RoboDK station: tarea2_isabellaceballos.rdk

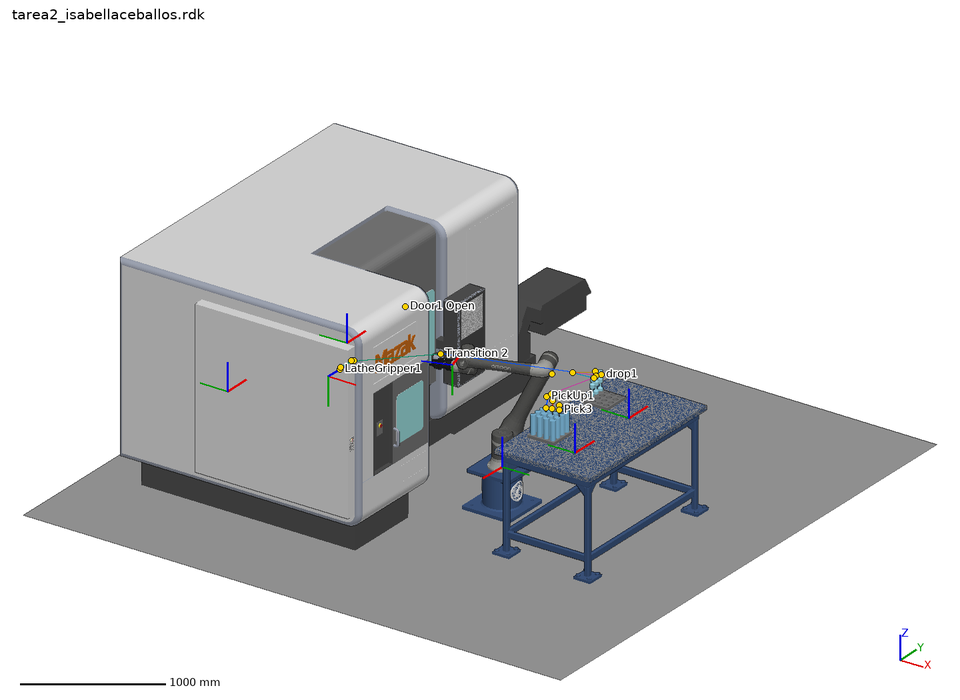
[picture v0: the station drawn from its stored meshes, robots at their saved joint values, targets as dots, program paths as lines]
Station tarea2_isabellaceballos (saved by RoboDK 5.5.1). Poses are relative to the parent item; angles as X-Y-Z fixed-axis rotations.
Station parameters (name, value as stored): TAGS, ['Machine Tending', 'CNC']
  - frame Omron TM12X Base at (300, 0, 70) mm, rotated rx 0 ry 0 rz -90 deg
    - robot Omron TM12X: 6 axes, payload 12 kg, reach 1300 mm, repeatability 0.1 mm, weight 33.3 kg
        modified DH rows (alpha deg, a mm, theta deg, d mm): 0, 0, 0, 165.2; 90, 0, 90, 0; 0, 636.1, 0, 0; 0, 557.9, -90, 156.3; -90, 0, 0, 106; 90, 0, 180, 113.15
        joint limits [-360, -360, -163, -360, -360, -360] to [360, 360, 163, 360, 360, 360]; home [0, 0, 90, -90, 90, 0]; saved at [291.3, -25.7, 113.76, -268.05, -85.72, 0]
      - frame RobotiQ HandE Dual Gripper at (0, 0, -5) mm
      - tool RobotiQ 2F-85 Gripper (Closed), TCP at (0, 0, 130) mm, size 134.4 x 157.6 x 75 mm
    - object Pedestal H12in (Type 1) at (0, 0, -300) mm, size 400 x 400 x 304.8 mm, geometry from Pedestal-H12in-Type-1.sld
  - frame Mazak Lathe Base at (-1000, 0, 650) mm, rotated rx 0 ry 0 rz 90 deg
    - frame Lathe at (-368.68, -104.77, -79.13) mm, rotated rx -90 ry 0 rz -90 deg
      - target LatheGripper1 (Cartesian target) at (-0.18, 0.1, 134.88) mm, rotated rx 0 ry 90 rz 165 deg; joints [296.712, 22.07, 84.693, -319.639, -67.09, 75.877] of Omron TM12X
      - target App1LatheGripper2 (Cartesian target) at (-0.18, 0.1, 301.9) mm, rotated rx 0 ry 90 rz 165 deg; joints [285.755, 19.624, 87.976, -318.559, -76.4, 81.971] of Omron TM12X
      - target App1LatheGripper (Cartesian target) at (-2.45, -8.35, 278.24) mm, rotated rx -90 ry -0.7 rz 75 deg; joints [284.667, 42.036, 44.196, -250.751, -75.843, 93.179] of Omron TM12X
      - target LatheGripper (Cartesian target) at (-2.58, -8.82, 147.35) mm, rotated rx -90 ry -0.7 rz 75 deg; joints [292.046, 45.075, 38.746, -247.697, -68.742, 95.287] of Omron TM12X
    - robot Mazak Lathe: 1 axes
        modified DH rows (alpha deg, a mm, theta deg, d mm): 0, 0, 0, 0 linear
        base shift (0, 0, 0) mm, rotated rx 0 ry 90 rz 0 deg
        joint limits [0] to [700]; home [0]; saved at [0]
  - frame Input at (1200, -410, 590) mm, rotated rx 0 ry 0 rz 90 deg
    - object Part Matrix at (0, 180, 30) mm, size 220 x 220 x 25 mm, geometry from Part Matrix.step
    - object Part 16 at (27.5, 207.5, 30) mm, size 40 x 40 x 150 mm, geometry from Part.step
    - object Part 15 at (27.5, 262.5, 30) mm, size 40 x 40 x 150 mm, geometry from Part.step
    - object Part 14 at (27.5, 317.5, 30) mm, size 40 x 40 x 150 mm, geometry from Part.step
    - object Part 12 at (82.5, 207.5, 30) mm, size 40 x 40 x 150 mm, geometry from Part.step
    - object Part 11 at (82.5, 262.5, 30) mm, size 40 x 40 x 150 mm, geometry from Part.step
    - object Part 10 at (82.5, 317.5, 30) mm, size 40 x 40 x 150 mm, geometry from Part.step
    - object Part 9 at (82.5, 372.5, 30) mm, size 40 x 40 x 150 mm, geometry from Part.step
    - object Part 8 at (137.5, 207.5, 30) mm, size 40 x 40 x 150 mm, geometry from Part.step
    - object Part 6 at (137.5, 317.5, 30) mm, size 40 x 40 x 150 mm, geometry from Part.step
    - object Part Done 16 at (27.5, 27.5, -20) mm, size 40.5 x 40.5 x 150 mm, geometry from Part Done.step
    - object Part Done 15 at (27.5, 82.5, -20) mm, size 40.5 x 40.5 x 150 mm, geometry from Part Done.step
    - object Part Done 14 at (27.5, 137.5, -20) mm, size 40.5 x 40.5 x 150 mm, geometry from Part Done.step
    - object Part Done 13 at (27.5, 192.5, -20) mm, size 40.5 x 40.5 x 150 mm, geometry from Part Done.step
    - object Part Done 12 at (82.5, 27.5, -20) mm, size 40.5 x 40.5 x 150 mm, geometry from Part Done.step
    - object Part Done 11 at (82.5, 82.5, -20) mm, size 40.5 x 40.5 x 150 mm, geometry from Part Done.step
    - object Part Done 10 at (82.5, 137.5, -20) mm, size 40.5 x 40.5 x 150 mm, geometry from Part Done.step
    - object Part Done 9 at (82.5, 192.5, -20) mm, size 40.5 x 40.5 x 150 mm, geometry from Part Done.step
    - object Part Done 8 at (137.5, 27.5, -20) mm, size 40.5 x 40.5 x 150 mm, geometry from Part Done.step
    - object Part Done 7 at (137.5, 82.5, -20) mm, size 40.5 x 40.5 x 150 mm, geometry from Part Done.step
    - object Part Done 6 at (137.5, 137.5, -20) mm, size 40.5 x 40.5 x 150 mm, geometry from Part Done.step
    - object Part Done 5 at (137.5, 192.5, -20) mm, size 40.5 x 40.5 x 150 mm, geometry from Part Done.step
    - object Part 7 at (137.5, 262.5, 30) mm, size 40 x 40 x 150 mm, geometry from Part.step
    - object Part 4 at (192.5, 207.5, 30) mm, rotated rx 0 ry 0 rz -180 deg, size 40 x 40 x 150 mm, geometry from Part.step
    - object Part Done 4 at (192.5, 27.5, -20) mm, rotated rx 0 ry 0 rz 180 deg, size 40.5 x 40.5 x 150 mm, geometry from Part Done.step
    - object Part 13 at (27.5, 372.5, 30) mm, size 40 x 40 x 150 mm, geometry from Part.step
    - target PickUp1 (Cartesian target) at (197.79, 377.57, 243.21) mm, rotated rx -90.01 ry 0 rz -179.05 deg; joints [78.517, -21.194, 99.72, -258.517, -102.431, -0.005] of Omron TM12X
    - target Pick1 (Cartesian target) at (192.26, 377.49, 159.76) mm, rotated rx -90.01 ry 0 rz -179.05 deg; joints [77.548, -21.82, 108.73, -266.901, -103.4, -0.006] of Omron TM12X
    - object Part 5 at (137.5, 372.5, 30) mm, size 40 x 40 x 150 mm, geometry from Part.step
    - target PickUp2 (Cartesian target) at (201.47, 332.43, 224.78) mm, rotated rx -90 ry 3.89 rz 135.95 deg; joints [107.585, -17.36, 99.274, -261.904, -28.363, 3.902] of Omron TM12X
    - target Pick2 (Cartesian target) at (194.9, 329.64, 168.72) mm, rotated rx -90 ry 3.89 rz 135.95 deg; joints [106.47, -17.482, 105.138, -267.647, -29.478, 3.901] of Omron TM12X
    - target PickUp3 (Cartesian target) at (198, 272.34, 206.6) mm, rotated rx -90.01 ry -0.01 rz 147.63 deg; joints [100.342, -14.09, 98.9, -264.802, -47.286, -0.002] of Omron TM12X
    - target Pick3 (Cartesian target) at (197.73, 271.91, 171.16) mm, rotated rx -90.01 ry -0.01 rz 147.63 deg; joints [100.293, -14.235, 102.652, -268.408, -47.336, -0.002] of Omron TM12X
  - frame Output at (1200, 230, 600) mm, rotated rx 0 ry 0 rz 90 deg
    - object Part Matrix at (0, 180, 30) mm, size 220 x 220 x 25 mm, geometry from Part Matrix.step
      - object Part 1 at (193.5, 178.91, -12.21) mm, rotated rx 0 ry -0.01 rz -111.33 deg, size 40 x 40 x 150 mm, geometry from Part.step
      - object Part Done 1 at (191.78, 194.55, 1.25) mm, rotated rx -0.18 ry -0.67 rz -15.38 deg, size 40.5 x 40.5 x 150 mm, geometry from Part Done.step
      - object Part 2 at (150.87, 185.46, -11.65) mm, rotated rx -2.71 ry -2.79 rz -101.16 deg, size 40 x 40 x 150 mm, geometry from Part.step
      - object Part Done 2 at (138.14, 192.48, 0.91) mm, rotated rx -0.17 ry -0.68 rz 49.72 deg, size 40.5 x 40.5 x 150 mm, geometry from Part Done.step
      - object Part 3 at (93.46, 178.8, -3.24) mm, rotated rx -4.21 ry 0.62 rz -139.81 deg, size 40 x 40 x 150 mm, geometry from Part.step
      - object Part Done 3 at (82.22, 190.38, 2.81) mm, rotated rx 4.03 ry 0 rz 22.82 deg, size 40.5 x 40.5 x 150 mm, geometry from Part Done.step
    - target drop1 (Cartesian target) at (198.5, 367.59, 147.55) mm, rotated rx -90 ry 0 rz 149.62 deg; joints [163.829, 5.576, 85.939, -271.515, 14.209, 0] of Omron TM12X
    - target UpDrop2 (Cartesian target) at (147.69, 382.37, 191.36) mm, rotated rx -90.01 ry 0 rz -145.27 deg; joints [150.104, -17.325, 101.671, -264.336, -64.625, 0.007] of Omron TM12X
    - target Drop2 (Cartesian target) at (147.19, 375.55, 157.21) mm, rotated rx -90.01 ry 0 rz -145.27 deg; joints [149.15, -17.018, 104.984, -267.956, -65.579, 0.007] of Omron TM12X
    - target Drop3 (Cartesian target) at (96.91, 360.44, 168.27) mm, rotated rx -93.89 ry -1.74 rz -172.1 deg; joints [156.377, -14.102, 122.108, -100.567, 31.62, 184.605] of Omron TM12X
  - frame World at (-2000, 0, 0) mm, rotated rx 0 ry 0 rz 90 deg
    - target Door1 Open (Cartesian target) at (700, -1000, 650) mm; joints [700, 0, 0, 0, 0, 0]
    - target Door1 Close (Cartesian target) at (0, -1000, 650) mm; joints [0, 0, 0, 0, 0, 0] of Mazak Lathe
    - object Floor at (250, -1940, -230) mm, size 4500 x 4500 x 0 mm, geometry from Floor (2).sld
    - object Table 1400x800x800mm at (-340, -3110, 590) mm, size 1420 x 820 x 800 mm, geometry from Table-1400x800x800mm.sld
    - target Home (Cartesian target) at (-159.05, -2821.45, 833.21) mm, rotated rx 0 ry 90 rz -134.05 deg; joints [118.439, -21.833, 100.089, -258.241, -17.509, 90.005] of Omron TM12X
    - target Transition1 (Cartesian target) at (332.55, -2486.73, 697.08) mm, rotated rx -89.14 ry -2.2 rz -141.74 deg; joints [240.5, -44.888, 123.151, -255.991, 22.223, -0.096] of Omron TM12X
    - target trans1 (Cartesian target) at (201.2, -2749.5, 833.2) mm, rotated rx 0 ry 90 rz -78.57 deg; joints [162.747, -30.859, 104.408, -253.528, -28.687, 90.017] of Omron TM12X
    - target Target 6 (Cartesian target) at (-159.05, -2821.45, 833.21) mm, rotated rx -116.03 ry 89.99 rz 109.92 deg; joints [120.666, -29.131, 103.705, -254.562, -60.282, 0.002] of Omron TM12X
    - target Transition 2 (joint target) at (110.77, -1705.81, 721.22) mm, rotated rx -130.72 ry 89.99 rz -68.7 deg; joints [291.3, -25.7, 113.76, -268.05, -85.72, 0]
    - target DOOROPEN (Cartesian target) at (700, -1000, 650) mm; joints [700] of Mazak Lathe
    - target DOOR CLOSE (Cartesian target) at (0, -1000, 650) mm; joints [0] of Mazak Lathe
    - target Target 10 (joint target) at (0, -1000, 650) mm; joints [0] of Mazak Lathe
  - folder Mechanism Programs
    - program OpenDoor1 (1 instructions, listed below)
    - program CloseDoor1 (1 instructions, listed below)
  - folder PickInput Programs
    - program Pick 1 (6 instructions, listed below)
    - program Pick 2 (6 instructions, listed below)
    - program Pick 3 (6 instructions, listed below)
  - folder DropOutput Programs
    - program Drop 1 (9 instructions, listed below)
    - program Drop 2 (8 instructions, listed below)
    - program Drop 3 (7 instructions, listed below)
  - folder Other Programs
    - program GoHome (3 instructions, listed below)
    - program ReplaceObjects (1 instructions, listed below)
    - program Init (6 instructions, listed below)
    - program PickLatheTransition (4 instructions, listed below)
  - folder Lath Programs
    - folder Work Programs
      - program Work 1 (3 instructions, listed below)
      - program Work 2 (3 instructions, listed below)
      - program Work 3 (3 instructions, listed below)
    - program PickLathe (11 instructions, listed below)
    - program DropLathe (10 instructions, listed below)
  - program Reset (2 instructions, listed below)
  - program MainProgram2 (22 instructions, listed below)
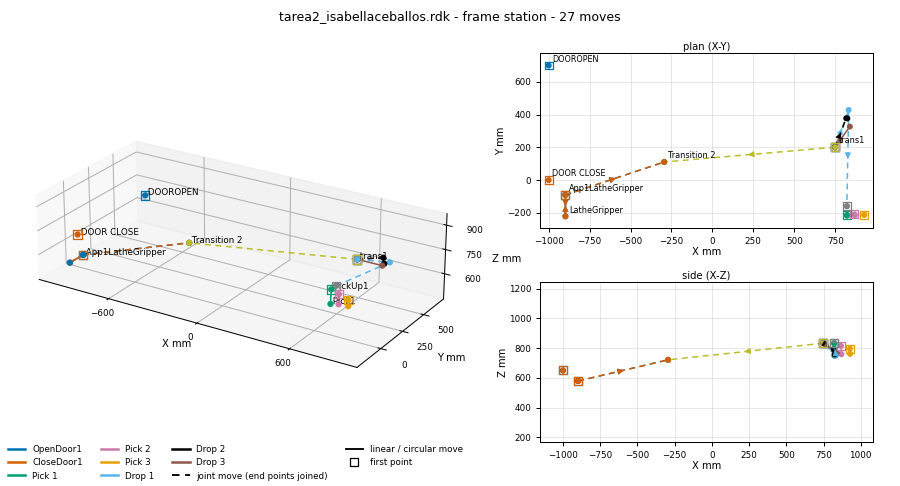
[picture p0: tool path of tarea2_isabellaceballos.rdk in frame station, 27 of 27 moves have a stored position in this frame; points joined in program order, loops and branches not executed]

--- program OpenDoor1 (robot Mazak Lathe) ---
  MoveJ (DOOROPEN)

--- program CloseDoor1 (robot Mazak Lathe) ---
  MoveJ (DOOR CLOSE)

--- program Pick 1 (robot Omron TM12X) ---
  Set Ref.: Input
  Est. herr: RobotiQ 2F-85 Gripper (Closed)
  MoveJ (PickUp1)
  MoveL (Pick1)
  Adjuntar a RobotiQ 2F-85 Gripper (Closed)
  Llamar GoHome

--- program Pick 2 (robot Omron TM12X) ---
  Set Ref.: Input
  Est. herr: RobotiQ 2F-85 Gripper (Closed)
  MoveJ (PickUp2)
  MoveL (Pick2)
  Adjuntar a RobotiQ 2F-85 Gripper (Closed)
  Llamar GoHome

--- program Pick 3 (robot Omron TM12X) ---
  Set Ref.: Input
  Est. herr: RobotiQ 2F-85 Gripper (Closed)
  MoveJ (PickUp3)
  MoveL (Pick3)
  Adjuntar a RobotiQ 2F-85 Gripper (Closed)
  Llamar GoHome

--- program Drop 1 (robot Omron TM12X) ---
  Set Ref.: World
  Est. herr: RobotiQ 2F-85 Gripper (Closed)
  MoveJ (trans1)
  Set Ref.: Output
  Est. herr: RobotiQ 2F-85 Gripper (Closed)
  MoveJ (drop1)
  Separar de RobotiQ 2F-85 Gripper (Closed)
  Set Ref.: World
  MoveJ (Home)

--- program Drop 2 (robot Omron TM12X) ---
  Set Ref.: World
  MoveJ (trans1)
  Set Ref.: Output
  Est. herr: RobotiQ 2F-85 Gripper (Closed)
  MoveJ (UpDrop2)
  MoveL (Drop2)
  Separar de RobotiQ 2F-85 Gripper (Closed)
  Llamar GoHome

--- program Drop 3 (robot Omron TM12X) ---
  Set Ref.: World
  MoveJ (trans1)
  Set Ref.: Output
  Est. herr: RobotiQ 2F-85 Gripper (Closed)
  MoveL (Target 4) -> target Drop3
  Separar de RobotiQ 2F-85 Gripper (Closed)
  Llamar GoHome

--- program GoHome (robot Omron TM12X) ---
  Set Ref.: World
  Set Tool: Gripper1 at (145, 0, 130) mm, rotated rx 45 ry 0 rz 90 deg
  MoveJ (Home)

--- program ReplaceObjects (robot Omron TM12X) ---
  Reemplazar objetos

--- program Init (robot Omron TM12X) ---
  Run OpenGripper1
  Run OpenGripper2
  Run CloseDoor1
  Run ReplaceObjects
  Show objects
  Hide objects

--- program PickLatheTransition (robot Omron TM12X) ---
  Set Ref.: World
  Set Tool: Gripper1 at (145, 0, 130) mm, rotated rx 45 ry 0 rz 90 deg
  MoveJ (trans1)
  MoveJ (Transition 2)

--- program Work 1 (robot Omron TM12X) ---
  Pausa 3.0 s
  Mostrar Part Done 1
  Hide Part 1

--- program Work 2 (robot Omron TM12X) ---
  Pausa 3.0 s
  Show Part Done 2
  Hide Part 2

--- program Work 3 (robot Omron TM12X) ---
  Pausa 3.0 s
  Show Part Done 3
  Hide Part 3

--- program PickLathe (robot Omron TM12X) ---
  Set Ref.: Lathe
  Est. herr: RobotiQ 2F-85 Gripper (Closed)
  Llamar OpenDoor1
  MoveJ (App1LatheGripper)
  MoveL (LatheGripper)
  Adjuntar a RobotiQ 2F-85 Gripper (Closed)
  Adjuntar a RobotiQ 2F-85 Gripper (Closed)
  MoveJ (App1LatheGripper)
  Set Ref.: World
  MoveJ (Transition 2)
  Llamar CloseDoor1

--- program DropLathe (robot Omron TM12X) ---
  Set Ref.: Lathe
  Est. herr: RobotiQ 2F-85 Gripper (Closed)
  Llamar OpenDoor1
  MoveJ (App1LatheGripper1)
  MoveL (LatheGripper)
  Separar de RobotiQ 2F-85 Gripper (Closed)
  MoveJ (App1LatheGripper1)
  Set Ref.: World
  MoveJ (Transition 2)
  Llamar CloseDoor1

--- program Reset (robot Omron TM12X) ---
  Call Init
  Call GoHome

--- program MainProgram2 (robot Omron TM12X) ---
  Llamar Init
  Llamar GoHome
  Llamar Pick 1
  Llamar PickLatheTransition
  Llamar DropLathe
  Llamar Work 1
  Llamar PickLathe
  Llamar Drop 1
  Llamar Pick 2
  Llamar PickLatheTransition
  Llamar DropLathe
  Llamar Work 2
  Reemplazar Part Done 2
  Llamar PickLathe
  Llamar Drop 2
  Llamar Pick 3
  Llamar PickLatheTransition
  Llamar DropLathe
  Llamar Work 3
  Reemplazar Part Done 3
  Llamar PickLathe
  Llamar Drop 3
